// TIA Portal V20 export
TYPE "typeDataToSafety"
// Information sent from the standard program to the safety program
// stored: Access Published, IsFailsafeCompliant true, Namespace Safety
   STRUCT
      ackSafetyFromHmi : Int;   // Acknowledge variable from operator control or monitoring system
      ackSafetyGlobal : Bool;   // Acknowledge command to ack all safety
      ackFromUnit1 : Bool;   // Acknowledge command coming from Unit 1
      ackSafetyFromMobileHMI : Bool;   // Acknowledge command coming from Mobile Panel
      resetSafetyFromMobileHMI : Bool;   // Reset command coming from Mobile Panel
      connectionBoxID_1 : Int;   // Mobile Panel Connection Box ID (extend list as needed)
      connectionBoxID_2 : Int;   // Mobile Panel Connection Box ID (extend list as needed)
      MobilePanelConnected : Bool;   // TRUE: connection box is connected
      MobilePanelPermissions : Bool;   // Transfer to Phmi Permissions
      DeselectBA10 : Bool;   // BA10 is not selected and no supply part
      DeselectBA15 : Bool;   // BA15 is not selected and no supply part
      DeselectBA40 : Bool;   // BA40 is not selected and no supply part
      DeselectBA60 : Bool;   // BA60 is not selected and no supply part
      PowerOnCommand : Bool;   // Power On Command
      InitializeEnable : Bool;
      BA060STOP : Bool;   // Stop Done For BA060 Request
      SepaGripperAxisXmoveToBa60 : Bool;
      unitMode : "Safety.typeUnitMode";   // Current mode of the unit
      BA060Mode : "Safety.typeUnitMode";
      unitState : "Safety.typeUnitStatus";   // Current States of the unit
      winderUsed : "Safety.typeWinderUseMode";
      StackDoor1 : "Safety.typeFdoorCommands";
      StackDoor2 : "Safety.typeFdoorCommands";
      StackDoor6 : "Safety.typeFdoorCommands";
      StackDoor7 : "Safety.typeFdoorCommands";
      scrapBox1Monitoring : "Safety.typeScrapBoxMonitoring";
      scrapBox2Monitoring : "Safety.typeScrapBoxMonitoring";
      hotWireCutterCmds : "Safety.typeHotWireCutter";
      clock : "Safety.typeGlobalClockMem";
      BrakeTest { S7_SetPoint := 'True'} : "Safety.typeBrakeTest";
   END_STRUCT;
   // // StackDoor1.Lock : zone1Fdoor1Lock
   // // StackDoor1.Unlock : zone1Fdoor1Unock
   // // StackDoor2.Lock : zone1Fdoor2Lock
   // // StackDoor2.Unlock : zone1Fdoor2Unock
   // // StackDoor6.Lock : zone1Fdoor6Lock
   // // StackDoor6.Unlock : zone1Fdoor6Unock
   // // StackDoor7.Lock : zone1Fdoor7Lock
   // // StackDoor7.Unlock : zone1Fdoor7Unock
END_TYPE
